// TIA Portal V15.1 export
// export: Created 2020-06-12T07:35:49.1474609Z, ExportSetting None, DisplayName Totally Integrated Automation Portal, DisplayVersion V15.1, DisplayName TIA Portal Openness, DisplayVersion V15.1, DisplayName STEP 7 Professional, DisplayVersion V15.1, DisplayName STEP 7 Safety, DisplayVersion V15.1, DisplayName WinCC Advanced, DisplayVersion V15.1
FUNCTION "HOOD_move" : Void   // FC851, FBD
TITLE = Hood Movement
{ S7_Optimized_Access := 'FALSE' }
// 15min dedusting ON because of argon
// stored: AutoNumber false, SetENOAutomatically False
   VAR_TEMP
      _no_pos : Bool;
      _lock_melt : Bool;
      _csf : Bool;
      _hod_up : Bool;
      _hod_dwn : Bool;
      _en_serv_dn : Bool;
      _seal_on : Bool;
      _ev06_on : Bool;
      _hd_dwn : Bool;
      _open_ev01 : Word;
      _close_ev01 : Word;
      tQ1 : Bool;
      tQ2 : Bool;
      tQ3 : Bool;
      tBypass : Bool;
      tBool : Bool;
   END_VAR
   VAR_TEMP   // added for the SCL form of the ladder/FBD networks
      _w1 : Bool;
      _w2 : Bool;
      _w3 : Bool;
   END_VAR
BEGIN

REGION Network 1: Common System Fault
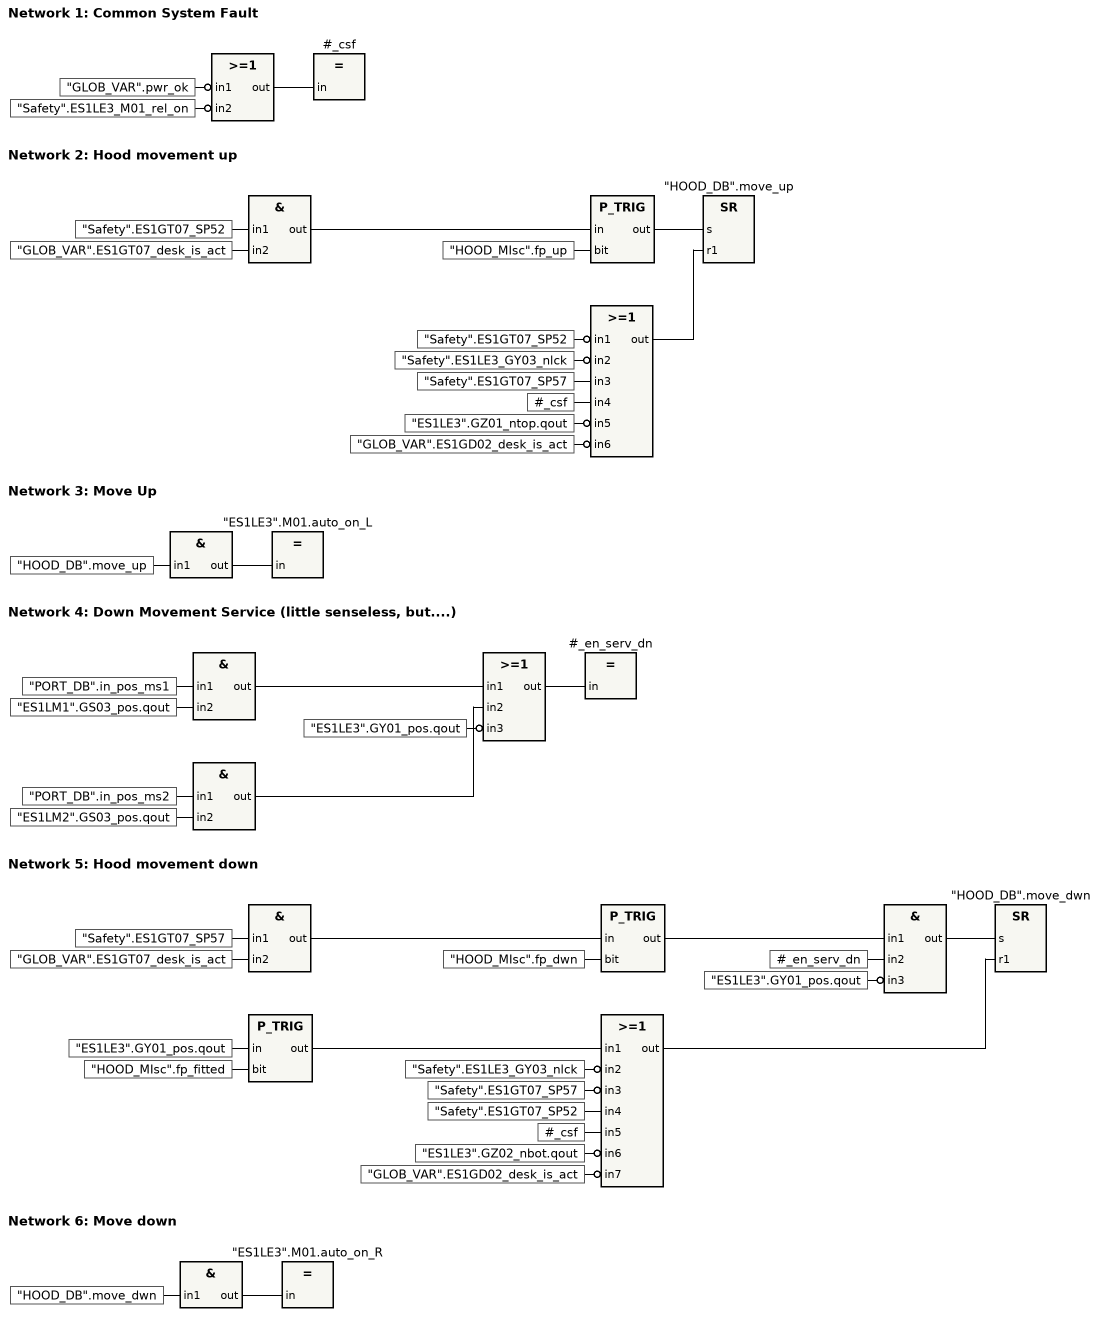
   #_csf := NOT "GLOB_VAR".pwr_ok OR NOT "Safety".ES1LE3_M01_rel_on;
END_REGION

REGION Network 2: Hood movement up
   #_w1 := "Safety".ES1GT07_SP52 AND "GLOB_VAR".ES1GT07_desk_is_act;
   #_w2 := #_w1 AND NOT "HOOD_MIsc".fp_up;   // rising edge
   "HOOD_MIsc".fp_up := #_w1;
   IF #_w2 THEN
       "HOOD_DB".move_up := TRUE;   // SR flip-flop
   END_IF;
   IF NOT "Safety".ES1GT07_SP52 OR NOT "Safety".ES1LE3_GY03_nlck OR "Safety".ES1GT07_SP57 OR #_csf OR NOT "ES1LE3".GZ01_ntop.qout OR NOT "GLOB_VAR".ES1GD02_desk_is_act THEN
       "HOOD_DB".move_up := FALSE;
   END_IF;
END_REGION

REGION Network 3: Move Up
   "ES1LE3".M01.auto_on_L := "HOOD_DB".move_up;
END_REGION

REGION Network 4: Down Movement Service (little senseless, but....)
   #_en_serv_dn := ("PORT_DB".in_pos_ms1 AND "ES1LM1".GS03_pos.qout) OR ("PORT_DB".in_pos_ms2 AND "ES1LM2".GS03_pos.qout) OR NOT "ES1LE3".GY01_pos.qout;
END_REGION

REGION Network 5: Hood movement down
   #_w1 := "Safety".ES1GT07_SP57 AND "GLOB_VAR".ES1GT07_desk_is_act;
   #_w2 := #_w1 AND NOT "HOOD_MIsc".fp_dwn;   // rising edge
   "HOOD_MIsc".fp_dwn := #_w1;
   #_w3 := "ES1LE3".GY01_pos.qout AND NOT "HOOD_MIsc".fp_fitted;   // rising edge
   "HOOD_MIsc".fp_fitted := "ES1LE3".GY01_pos.qout;
   IF #_w2 AND #_en_serv_dn AND NOT "ES1LE3".GY01_pos.qout THEN
       "HOOD_DB".move_dwn := TRUE;   // SR flip-flop
   END_IF;
   IF #_w3 OR NOT "Safety".ES1LE3_GY03_nlck OR NOT "Safety".ES1GT07_SP57 OR "Safety".ES1GT07_SP52 OR #_csf OR NOT "ES1LE3".GZ02_nbot.qout OR NOT "GLOB_VAR".ES1GD02_desk_is_act THEN
       "HOOD_DB".move_dwn := FALSE;
   END_IF;
END_REGION

REGION Network 6: Move down
   "ES1LE3".M01.auto_on_R := "HOOD_DB".move_dwn;
END_REGION

REGION Network 7: handover setpoint
   // 7.500000e+001
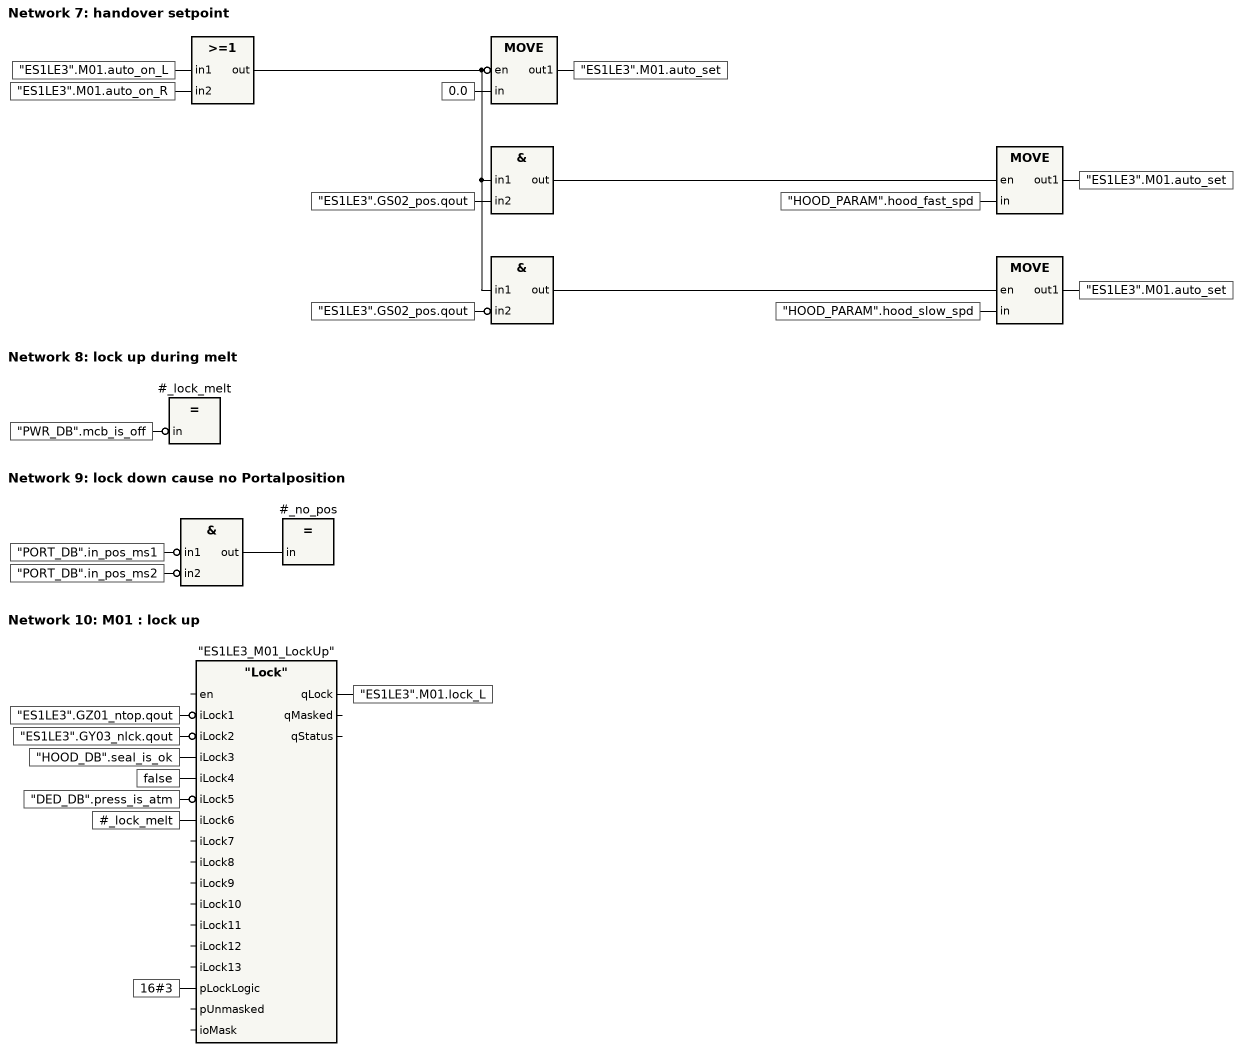
   #_w1 := "ES1LE3".M01.auto_on_L OR "ES1LE3".M01.auto_on_R;
   IF NOT #_w1 THEN "ES1LE3".M01.auto_set := 0.0; END_IF;
   IF #_w1 AND "ES1LE3".GS02_pos.qout THEN "ES1LE3".M01.auto_set := "HOOD_PARAM".hood_fast_spd; END_IF;
   IF #_w1 AND NOT "ES1LE3".GS02_pos.qout THEN "ES1LE3".M01.auto_set := "HOOD_PARAM".hood_slow_spd; END_IF;
END_REGION

REGION Network 8: lock up during melt
   #_lock_melt := NOT "PWR_DB".mcb_is_off;
END_REGION

REGION Network 9: lock down cause no Portalposition
   #_no_pos := NOT "PORT_DB".in_pos_ms1 AND NOT "PORT_DB".in_pos_ms2;
END_REGION

REGION Network 10: M01 : lock up
   "ES1LE3_M01_LockUp"(iLock1 := NOT "ES1LE3".GZ01_ntop.qout,   // "Lock"
                       iLock2 := NOT "ES1LE3".GY03_nlck.qout,
                       iLock3 := "HOOD_DB".seal_is_ok,
                       iLock4 := false,
                       iLock5 := NOT "DED_DB".press_is_atm,
                       iLock6 := #_lock_melt,
                       pLockLogic := 16#3,
                       qLock => "ES1LE3".M01.lock_L);
END_REGION

REGION Network 11: M01 : lock down
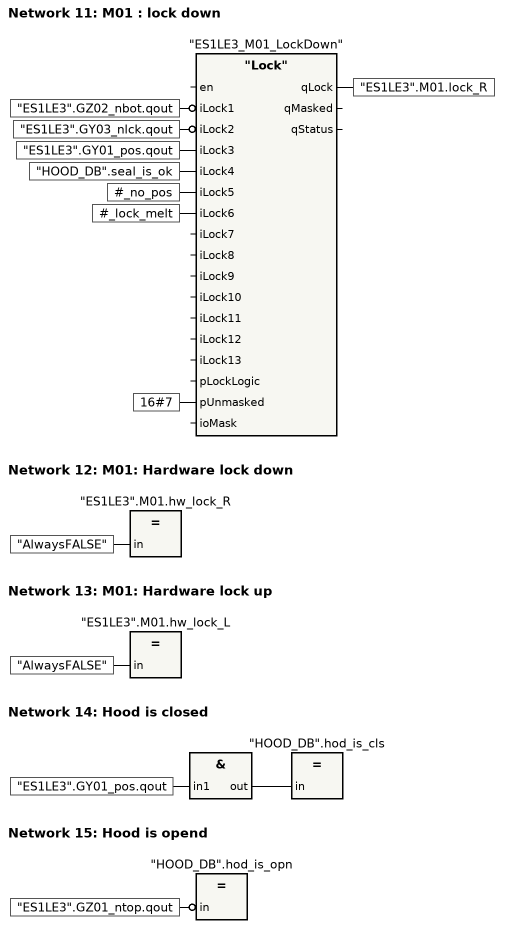
   "ES1LE3_M01_LockDown"(iLock1 := NOT "ES1LE3".GZ02_nbot.qout,   // "Lock"
                         iLock2 := NOT "ES1LE3".GY03_nlck.qout,
                         iLock3 := "ES1LE3".GY01_pos.qout,
                         iLock4 := "HOOD_DB".seal_is_ok,
                         iLock5 := #_no_pos,
                         iLock6 := #_lock_melt,
                         pUnmasked := 16#7,
                         qLock => "ES1LE3".M01.lock_R);
END_REGION

REGION Network 12: M01: Hardware lock down
   "ES1LE3".M01.hw_lock_R := "AlwaysFALSE";
END_REGION

REGION Network 13: M01: Hardware lock up
   "ES1LE3".M01.hw_lock_L := "AlwaysFALSE";
END_REGION

REGION Network 14: Hood is closed
   "HOOD_DB".hod_is_cls := "ES1LE3".GY01_pos.qout;
END_REGION

REGION Network 15: Hood is opend
   "HOOD_DB".hod_is_opn := NOT "ES1LE3".GZ01_ntop.qout;
END_REGION
END_FUNCTION
